INTERFACE I_Mc3MotionTaskCollection EXTENDS I_TaskResult

METHOD AddTask
VAR_INPUT
	Task : I_Mc3MotionTask;
END_VAR
END_METHOD

{attribute 'monitoring' := 'call'}
PROPERTY ErrorTask : T_MaxString
GET
END_GET
END_PROPERTY

METHOD RemoveTaskByInstance
VAR_INPUT
	Task : I_Mc3MotionTask;
END_VAR
END_METHOD

END_INTERFACE

(* stored: Version 1.1.0.1, ProductVersion 3.1.4026.20
   Itf I_Mc3MotionTaskCollection: Id {0693867d-01b1-4609-bc6c-ec0ff4adb1dd}
   Method AddTask: Id {c9cc9289-4428-46a4-9845-934b2dc5e811}
   Property ErrorTask: Id {e7dce802-b9c8-478f-aa81-d236b24591e5}
   Get Get: Id {40026c20-b501-4d34-a1f5-a9830732a826}
   Method RemoveTaskByInstance: Id {04b332a2-0867-42de-88ea-293be0fc1a3d} *)
